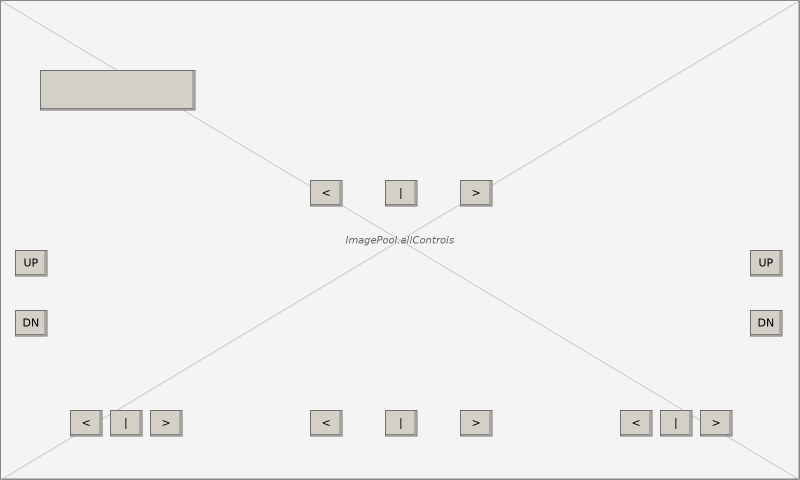
VISUALIZATION allControls  // 800x480
    Image (0,0 800x480), image: ImagePool.allControls
    Button (700,410 32x26), ">"
        OnMouseClick: execute { rightBelt(1); }
    Button (620,410 32x26), "<"
        OnMouseClick: execute { rightBelt(2); }
    Button (460,410 32x26), ">"
        OnMouseClick: execute { bottomBelt(1); }
    Button (310,410 32x26), "<"
        OnMouseClick: execute { bottomBelt(2); }
    Button (150,410 32x26), ">"
        OnMouseClick: execute { leftBelt(1); }
    Button (70,410 32x26), "<"
        OnMouseClick: execute { leftBelt(2); }
    Button (750,310 32x26), "DN"
        OnMouseClick: execute { rightLift(4); }
    Button (750,250 32x26), "UP"
        OnMouseClick: execute { rightLift(3); }
    Button (15,250 32x26), "UP"
        OnMouseClick: execute { leftLift(3); }
    Button (15,310 32x26), "DN"
        OnMouseClick: execute { leftLift(4); }
    Button (460,180 32x26), ">"
        OnMouseClick: execute { topBelt(1); }
    Button (310,180 32x26), "<"
        OnMouseClick: execute { topBelt(2); }
    Button (40,70 155x40), image: Buttons.homeButton
        OnMouseDown: change screen: Main
        OnMouseDown: execute { MAIN.allControls:=FALSE; }
    Button (110,410 32x26), "|"
        OnMouseClick: execute { leftBelt(0); }
    Button (385,410 32x26), "|"
        OnMouseClick: execute { bottomBelt(0); }
    Button (660,410 32x26), "|"
        OnMouseClick: execute { rightBelt(0); }
    Button (385,180 32x26), "|"
        OnMouseClick: execute { topBelt(0); }
END_VISUALIZATION

(* stored: Version 1.1.0.1, ProductVersion 3.1.4018.2
   Visu allControls: Id {cfda31ca-405c-4c7a-b47a-1f1d0c909d29} *)
